// Mitsubishi GX Works2 project: LRI - PLC - SEM ST V1   PLC: Q03UDV

// task Task_01 (event TRUE, interval 0, priority 31): POU_01

PROGRAM POU_01
VAR
  x_EstadosSemafaros : ARRAY [0..9] OF BOOL;
  st_Semafora_1 : st_Semafora;
END_VAR



st_Semafora_1(i_AtivarSemaforo:= 1 ,o_Verde1:= x_EstadosSemafaros[0] ,o_Amarelo1:= x_EstadosSemafaros[1] ,o_Vermelho1:= x_EstadosSemafaros[2] ,o_Verde2:= x_EstadosSemafaros[3] ,
	o_Amarelo2:= x_EstadosSemafaros[4] ,o_Vermelho2:= x_EstadosSemafaros[5] );
END_PROGRAM

FUNCTION_BLOCK st_Semafora
VAR_INPUT
  i_AtivarSemaforo : BOOL;
END_VAR
VAR_OUTPUT
  o_Verde1 : BOOL;
  o_Amarelo1 : BOOL;
  o_Vermelho1 : BOOL;
  o_Verde2 : BOOL;
  o_Amarelo2 : BOOL;
  o_Vermelho2 : BOOL;
END_VAR
VAR
  x_Time1 : BOOL;
  x_Time2 : BOOL;
END_VAR


OUT_T(i_AtivarSemaforo,TC1,100);
OUT(TS1,x_Time1);

IF x_Time1 >= 0 THEN
	o_Verde1 := 0;
	o_Vermelho2 := 0;
END_IF;
END_FUNCTION_BLOCK
